Staubli VAL3: start.pgx

public program start()
begin
  call Main(0)
end
